TYPE ST_MultiLeaderMotionCoupling :
STRUCT
    {attribute 'pytmc' := '
        pv: bEnable
        io: io
        field: DESC Set and hold TRUE to allow the axis to run in multi-leader mode.
    '}
    bEnable: BOOL;

    {attribute 'pytmc' := '
        pv: bReset
        io: io
        field: DESC Set and release TRUE to fully reset errors and state machine.
    '}
    bReset: BOOL;

    {attribute 'pytmc' := '
        pv: bBusy
        io: i
        field: DESC TRUE indicates state machine running and not in error state.
    '}
    bBusy: BOOL;

    {attribute 'pytmc' := '
        pv: sStatusMsg
        io: i
        field: DESC String used to give helpful messages.
    '}
    sStatusMsg: T_MaxString;

    // Ex: TIID^Device 2 (EtherCAT)^B950-233-WALL-S-R01-DRL-01^EL7047_02_11^STM Status^Status^Ready
    {attribute 'pytmc' := '
        pv: bFollowerDriveReady
        io: i
        field: DESC Linked to the ready status of the drive.
    '}
    bFollowerDriveReady AT %I*: BOOL; // Link to the ready status of the drive

    {attribute 'pytmc' := '
        pv: bUseDynamicLimits
        io: io
        field: DESC Set AND hold TRUE to enable dynamic limits to acc, vel, AND pos.
    '}
    bUseDynamicLimits: BOOL;

    {attribute 'pytmc' := '
        pv: fTargetAcc
        io: io
        field: DESC The target acceleration.
    '}
    fTargetAcc: LREAL; // Set in software to allow axis to target an acceleration based on multiple leaders.

    {attribute 'pytmc' := '
        pv: fTargetVel
        io: io
        field: DESC The target velocity.
    '}
    fTargetVel: LREAL; // Set in software to allow axis to target a velocity based on multiple leaders.

    {attribute 'pytmc' := '
        pv: fTargetPos
        io: io
        field: DESC The target position.
    '}
    fTargetPos: LREAL; // Set in software to allow axis to target a position based on multiple leaders.

    {attribute 'pytmc' := '
        pv: fPosDelta
        io: i
        field: DESC Target position minus position.
    '}
    fPosDelta : LREAL; // Difference between current position and target position.

    {attribute 'pytmc' := '
        pv: fTTGain
        io: io
        field: DESC Target tracking gain.
    '}
    fTargetTrackingGain: LREAL := 1; // Gain used to tune target tracking when within target position window.

    {attribute 'pytmc' := '
        pv: fHaltPos
        io: i
        field: DESC Position at which axis halted.
    '}
    fHaltPos: LREAL; // Position at which halt is called. Allows for centering deadband.

    {attribute 'pytmc' := 'pv: stAcc'}
    stAcc: ST_BoundedValue;

    {attribute 'pytmc' := 'pv: stVel'}
    stVel: ST_BoundedValue;

    {attribute 'pytmc' := 'pv: stPos'}
    stPos: ST_BoundedValue;

    {attribute 'pytmc' := '
        pv: nDir
        io: i
        field: DESC Internally calculated direction value for external setpoint generator.
    '}
    nDir: DINT;

    {attribute 'pytmc' := '
        pv: bError
        io: i
        field: DESC TRUE if an error is active.
    '}
    bError: BOOL;

    {attribute 'pytmc' := '
        pv: sErrorMsg
        io: i
        field: DESC Displays error message relevant to the active error. Empty otherwise.
    '}
    sErrorMsg: T_MaxString;

    {attribute 'pytmc' := '
        pv: sErrorHelp
        io: i
        field: DESC Displays additional help for the active rror. Empty otherwise.
    '}
    sErrorHelp: T_MaxString;

    {attribute 'pytmc' := '
        pv: eState
        io: i
        field: DESC Records the current state of the multi-leader function block.
    '}
    eState: E_MultiLeaderMotionCoupling;
END_STRUCT
END_TYPE

(* stored: Version 1.1.0.1
   DUT ST_MultiLeaderMotionCoupling: Id {3deae775-0f2c-41fa-8a74-ef3b2b206a82} *)
